FUNCTION_BLOCK FB_System_MVKW_100
VAR_INPUT
	Freigabe_auto				: BOOL;
	Freigabe_Deakt_auto			: BOOL;
	Betrieb_Anford_auto			: BOOL;
END_VAR
VAR_OUTPUT
	{attribute 'OPC.UA.DA' := '1'}Steuerung					: ST_System_MVKW_Steuerung;		
	{attribute 'OPC.UA.DA' := '1'}Stellwert					: ST_System_MVKW_Stellwert;		
	{attribute 'OPC.UA.DA' := '1'}Zustand						: ST_System_MVKW_Zustand;	
	{attribute 'OPC.UA.DA' := '1'}Parameter					: ST_System_MVKW_Parameter;		
END_VAR
VAR
	Pumpe_100							: FB_PU;
	Stellventil_100						: FB_SV;
	Maschinenversorgung_EMAG_GT	: FB_MV_EMAG_GT;

	Zustandscheck						: FB_System_MVKW_Zustandscheck;
	Logik								: FB_System_MVKW_Logik;
	Ablaufsteuerung						: FB_System_MVKW_Ablaufsteuerung;


	Maschinenversorgung_HD				: FB_MV_HD;
END_VAR
VAR // added by the converter: edge detectors and wires of the graphical bodies
    _w1 : ANY;
END_VAR

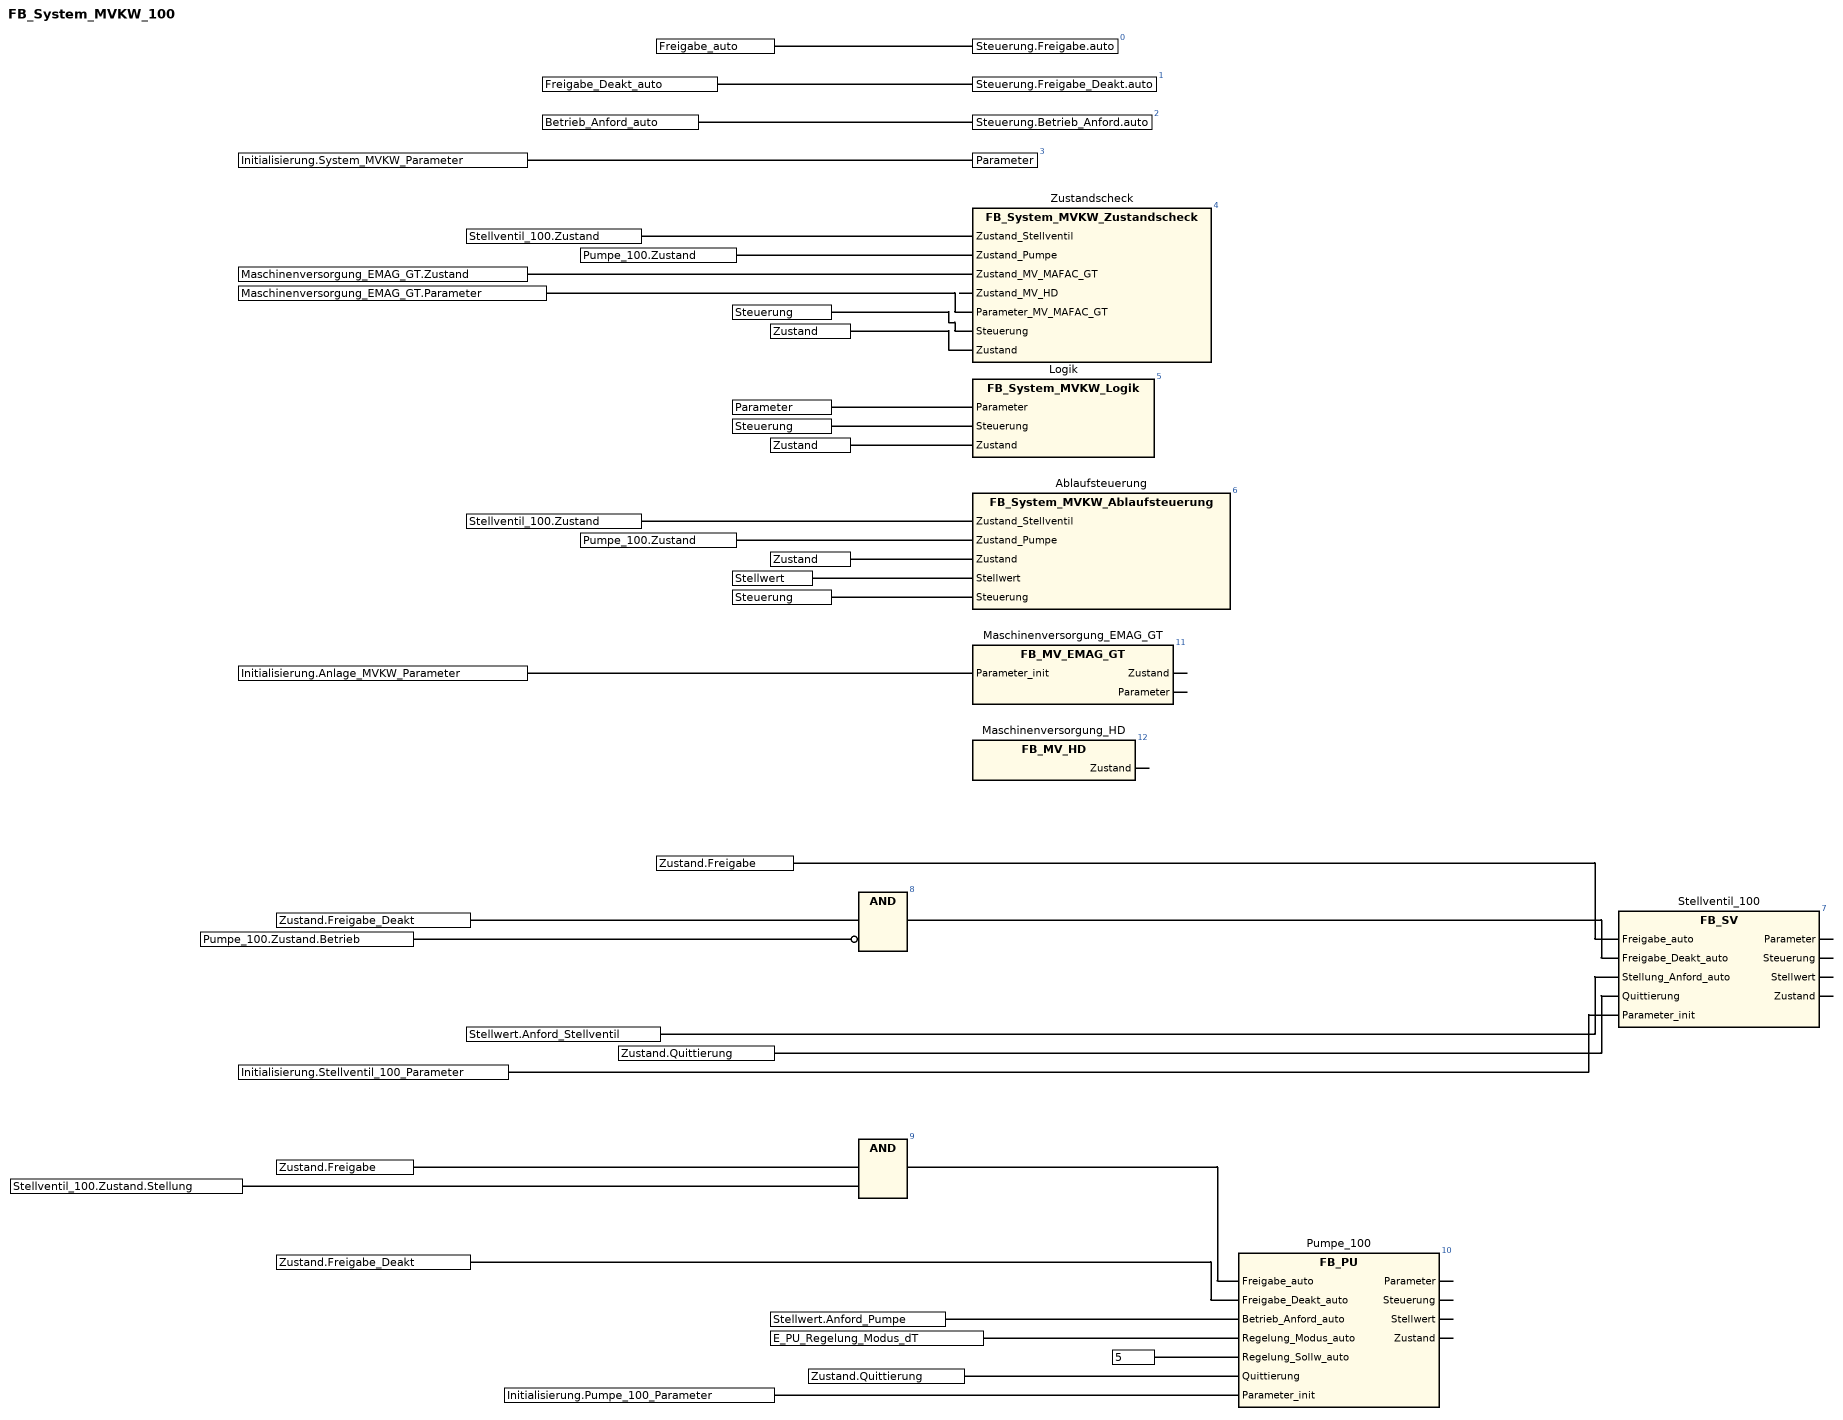
Steuerung.Freigabe.auto := Freigabe_auto;
Steuerung.Freigabe_Deakt.auto := Freigabe_Deakt_auto;
Steuerung.Betrieb_Anford.auto := Betrieb_Anford_auto;
Parameter := Initialisierung.System_MVKW_Parameter;
Zustandscheck(
    Zustand_Stellventil := Stellventil_100.Zustand,
    Zustand_Pumpe := Pumpe_100.Zustand,
    Zustand_MV_MAFAC_GT := Maschinenversorgung_EMAG_GT.Zustand,
    Parameter_MV_MAFAC_GT := Maschinenversorgung_EMAG_GT.Parameter,
    Steuerung := Steuerung,
    Zustand := Zustand); // FB_System_MVKW_Zustandscheck
Logik(Parameter := Parameter, Steuerung := Steuerung, Zustand := Zustand); // FB_System_MVKW_Logik
Ablaufsteuerung(
    Zustand_Stellventil := Stellventil_100.Zustand,
    Zustand_Pumpe := Pumpe_100.Zustand,
    Zustand := Zustand,
    Stellwert := Stellwert,
    Steuerung := Steuerung); // FB_System_MVKW_Ablaufsteuerung
Stellventil_100(
    Freigabe_auto := Zustand.Freigabe,
    Freigabe_Deakt_auto := _w1,
    Stellung_Anford_auto := Stellwert.Anford_Stellventil,
    Quittierung := Zustand.Quittierung,
    Parameter_init := Initialisierung.Stellventil_100_Parameter); // FB_SV
_w1 := Zustand.Freigabe_Deakt AND NOT Pumpe_100.Zustand.Betrieb;
Pumpe_100(
    Freigabe_auto := Zustand.Freigabe AND Stellventil_100.Zustand.Stellung,
    Freigabe_Deakt_auto := Zustand.Freigabe_Deakt,
    Betrieb_Anford_auto := Stellwert.Anford_Pumpe,
    Regelung_Modus_auto := E_PU_Regelung_Modus_dT,
    Regelung_Sollw_auto := 5,
    Quittierung := Zustand.Quittierung,
    Parameter_init := Initialisierung.Pumpe_100_Parameter); // FB_PU
Maschinenversorgung_EMAG_GT(Parameter_init := Initialisierung.Anlage_MVKW_Parameter); // FB_MV_EMAG_GT
Maschinenversorgung_HD(); // FB_MV_HD

END_FUNCTION_BLOCK

(* stored: Version 1.1.0.1, ProductVersion 3.1.4024.9
   POU FB_System_MVKW_100: Id {baf259c5-7603-4c7a-89d6-a7978f74b82f}, SpecialFunc None *)
